// TIA Portal V20 export
// export: Created 2025-12-01T14:56:13.844196Z, ExportSetting None, DisplayName Totally Integrated Automation Portal, DisplayVersion V20 Update 3, DisplayName TIA Portal Openness, DisplayVersion V20 Update 3, DisplayName TIA Portal Version Control Interface, DisplayVersion V20 Update 3, DisplayName STEP 7 Professional, DisplayVersion V20 Update 3, DisplayName STEP 7 Safety, DisplayVersion V20 Update 2, DisplayName WinCC Basic/Comfort/Advanced, DisplayVersion V20 Update 3, DisplayName WinCC Professional, DisplayVersion V20 Update 3, DisplayName WinCC Unified, DisplayVersion V20 Update 3
TYPE "UDT_DatosDispositivoMaquina"
   STRUCT
      EstadoRecepcionEvento : UInt;   // Estado de la recepcion del Evento
      EstadoEmisionEvento : UInt;   // Estado de la Emision del Evento
      EstadoGeneralEvento : UInt;   // Estado general de los Eventos (Peticiones)
      EstadoOrdenDispo : UInt;   // Estado de la Orden enviada al Dispositivo
      EstadoPresenciaDispo : UInt;   // Estaod de la Presencia enviada del Dispositivo
      TMP_Reset : UDInt;   // Temporizador para Fin Reset
      TMP_ParoBlando : UDInt;   // Temporizador para Fin Paro Blando
      Prioridad : UInt;   // Prioridad del Dispositivo
      StatusActual : Word;   // Status actual del Dispositivo (Ultimo Evento)
      ErrorActual : UDInt;   // Error Actual del Dispositivo (Ultimo Evento)
      StatusReal : Word;   // Status Real del Dispositivo
      ErrorReal : UDInt;   // Error Real del Dispositivo
      MemoriaEstado : UInt;   // Nuevo Status de Estado de Trabajo de la Maquina
      Operacion : UInt;   // Cambio Status de Estado de Trabajo de la Maquina
      Memorias : Struct   // Memorizacion de los Flancos de cambio de estado
         MFL_Marcha : Bool;
         MFL_Paro : Bool;
         MFL_Reset : Bool;
         MFL_Auto : Bool;
         MFL_Remoto : Bool;
         MFL_Manual : Bool;
         MFL_ParoBlando : Bool;
         DesHabilitado : Bool;
      END_STRUCT;
      VTD_ELEV : Struct
         Operacion : UInt;
         Respuesta : UInt;
         MesaHorquilla : UInt;
         MesaCargaDesCarga : UInt;
      END_STRUCT;
   END_STRUCT;
END_TYPE
